{attribute addProperty BoxType "EL6751--0000"}
{attribute addProperty Id "InfoDataInfoData_275E336312816"}
{attribute addProperty CRC "2358898256"}
{attribute addProperty SizeInBites "128"}
{attribute addProperty SizeInBytes "16"}
TYPE EL6751_8C99EE50 :
STRUCT
	{attribute addProperty Name "InfoData"}
	InfoData : InfoData_275E3363;
END_STRUCT
END_TYPE

(* stored: Version 1.2.0.0, ProductVersion 3.1.4024.9
   DUT EL6751_8C99EE50: Id {5912a19b-2716-4931-9370-4d4a26d8f6c6} *)
